# EPICS IOC start-up script: iocsh/ethercatmcPTP.iocsh
dbLoadRecords("ethercatmcPTP.template", "PREFIX=$(PREFIX), MOTOR_PORT=$(MOTOR_PORT)")
